// TIA Portal V15.1 export
// export: Created 2024-05-17T05:38:32.5503096Z, ExportSetting WithDefaults, DisplayName Totally Integrated Automation Portal, DisplayVersion V15.1 Update 5, DisplayName TIA Portal Openness, DisplayVersion V15.1 Update 5, DisplayName SINAMICS Startdrive Advanced, DisplayVersion V15.1, DisplayName G130, G150, S120, S150, SINAMICS MV, S210, DisplayVersion V15.1, DisplayName G110M, G120, G120C, G120D, G120P, DisplayVersion V15.1, DisplayName STEP 7 Professional, DisplayVersion V15.1 Update 5, DisplayName STEP 7 Safety, DisplayVersion V15.1, DisplayName WinCC Professional, DisplayVersion V15.1 Update 5, DisplayName SIMATIC Visualization Architect, DisplayVersion V15.1
FUNCTION_BLOCK "LMovFnc3Pos"   // FB2187, FBD
TITLE = LMovFnc3Pos
{ S7_Optimized_Access := 'TRUE' }
AUTHOR : VCC
FAMILY : Tooling
VERSION : 0.1
// =============================================================================
// This module will be used for the steering of a three Position movement.
// It will get the commands from different Modes, evaluate the status of the 
// Interlock and give the command to the Actuator or direct to simple outputs.
// =============================================================================
// stored: AutoNumber false, IsIECCheckEnabled false, IsRetainMemResEnabled false, MemoryReserve 100, SetENOAutomatically False, UDAEnableTagReadback false
   VAR_INPUT
      I_Pos1 { ExternalAccessible := 'False'; ExternalVisible := 'False'; ExternalWritable := 'False'} : Bool;   // Position Set detection or summary / Position 1 Detection
      I_Pos2 { ExternalAccessible := 'False'; ExternalVisible := 'False'; ExternalWritable := 'False'} : Bool;   // Position 2 Detection
      I_Pos3 { ExternalAccessible := 'False'; ExternalVisible := 'False'; ExternalWritable := 'False'} : Bool;   // Position Reset detection or summary / Position 3 Detection
      I_PBSet { ExternalAccessible := 'False'; ExternalVisible := 'False'; ExternalWritable := 'False'} : Bool;   // Push button for Set direction (used in manual with button OP panels )
      I_PBReset { ExternalAccessible := 'False'; ExternalVisible := 'False'; ExternalWritable := 'False'} : Bool;   // Push button for reset direcion (used in manual with pushbutton OP panels) / Push button for Reset direction (used in manual with Pushbutton OP panels)
      I_Pos1Begin { ExternalAccessible := 'False'; ExternalVisible := 'False'; ExternalWritable := 'False'} : Bool;   // Function Set begin selection / Function Pos1 begin selection
      I_Pos2Begin { ExternalAccessible := 'False'; ExternalVisible := 'False'; ExternalWritable := 'False'} : Bool;   // Function Set begin selection / Function Pos2 begin selection
      I_Pos3Begin { ExternalAccessible := 'False'; ExternalVisible := 'False'; ExternalWritable := 'False'} : Bool;   // Function Reset begin selection / Function Pos3 begin selection
      I_Pos1IntlkOK { ExternalAccessible := 'False'; ExternalVisible := 'False'; ExternalWritable := 'False'} : Bool;   // Set Interlock / Pos1 Interlock
      I_Pos2IntlkOK { ExternalAccessible := 'False'; ExternalVisible := 'False'; ExternalWritable := 'False'} : Bool;   // Set Interlock / Pos2 Interlock
      I_Pos3IntlkOK { ExternalAccessible := 'False'; ExternalVisible := 'False'; ExternalWritable := 'False'} : Bool;   // Reset Interlock / Pos3 Interlock
      I_MiddleReachedManSTOP { ExternalAccessible := 'False'; ExternalVisible := 'False'; ExternalWritable := 'False'} : Bool;   // Middle pos reached
      I_SafetyOk { ExternalAccessible := 'False'; ExternalVisible := 'False'; ExternalWritable := 'False'} : Bool;   // Safety Ok
      I_HardwareOk { ExternalAccessible := 'False'; ExternalVisible := 'False'; ExternalWritable := 'False'} : Bool;   // Safety Ok / Hardware Ok
   END_VAR
   VAR_OUTPUT
      O_CmdPos1 { ExternalAccessible := 'False'; ExternalVisible := 'False'; ExternalWritable := 'False'} : Bool;   // Command to activate Set movement / Command to Activate Pos1 movement
      O_CmdPos2 { ExternalAccessible := 'False'; ExternalVisible := 'False'; ExternalWritable := 'False'} : Bool;   // Command to activate Set movement / Command to Activate Pos2 movement
      O_CmdPos3 { ExternalAccessible := 'False'; ExternalVisible := 'False'; ExternalWritable := 'False'} : Bool;   // Command to activate Reset movement / Command to Activate Pos3 movement
      O_FuncRunning { ExternalAccessible := 'False'; ExternalVisible := 'False'; ExternalWritable := 'False'} : Bool;   // Signal that the function is running
      O_FuncBusyTM { ExternalAccessible := 'False'; ExternalVisible := 'False'; ExternalWritable := 'False'} : Bool;   // Memory Signal that the function is busy
      O_Pos1Finished { ExternalAccessible := 'False'; ExternalVisible := 'False'; ExternalWritable := 'False'} : Bool;   // Function Set finished to Master Sequencing / Function Pos1 finished to Master Sequencing
      O_Pos2Finished { ExternalAccessible := 'False'; ExternalVisible := 'False'; ExternalWritable := 'False'} : Bool;   // Function Set finished to Master Sequencing / Function Pos2 finished to Master Sequencing
      O_Pos3Finished { ExternalAccessible := 'False'; ExternalVisible := 'False'; ExternalWritable := 'False'} : Bool;   // Function Reset finished to Master Sequencing / Function Pos3 finished to Master Sequencing
      O_IntlkPos1Alm { ExternalAccessible := 'False'; ExternalVisible := 'False'; ExternalWritable := 'False'} : Bool;   // Alarm interlock Set / Alarm Interlock Pos1
      O_IntlkPos2Alm { ExternalAccessible := 'False'; ExternalVisible := 'False'; ExternalWritable := 'False'} : Bool;   // Alarm interlock Set / Alarm Interlock Pos2
      O_IntlkPos3Alm { ExternalAccessible := 'False'; ExternalVisible := 'False'; ExternalWritable := 'False'} : Bool;   // Alarm interlock Reset / Alarm Interlock Reset
      O_FuncIsSelInMan { ExternalAccessible := 'False'; ExternalVisible := 'False'; ExternalWritable := 'False'} : Bool;   // The function is selected in manual mode / The function is Selected in manual Mode
      O_LED { ExternalAccessible := 'False'; ExternalVisible := 'False'; ExternalWritable := 'False'} : Bool;   // LED - Indication
      O_AlarmABCondition { ExternalAccessible := 'False'; ExternalVisible := 'False'; ExternalWritable := 'False'} : Bool;   // Alarms AB condition / Alarm AB Condition
   END_VAR
   VAR_IN_OUT
      IO_Modes : "Modes";   // Modes
      H_HMI : "H_HMI";   // Animation
      H_MovFnc3Pos : "H_MovFnc3Pos";   // Animation
      H_FncSelInHMI { ExternalAccessible := 'False'; ExternalVisible := 'False'; ExternalWritable := 'False'} : Bool;   // This function is selected to run from HMI / This function is Selected to run from HMI
      C_AlarmResetUsed { ExternalAccessible := 'False'; ExternalVisible := 'False'; ExternalWritable := 'False'} : Bool;   // If true, the alrms will be stored untill reseted / If TRUE The Alarms will be stored untill Reseted
      C_EnableMemBegin { ExternalAccessible := 'False'; ExternalVisible := 'False'; ExternalWritable := 'False'} : Bool;   // Enable memory Begin (Command request is memorised until pos reached) / Enable memory Begin (Command Request is memorised until pos reached)
      C_EnIntlkAlm { ExternalAccessible := 'False'; ExternalVisible := 'False'; ExternalWritable := 'False'} : Bool := TRUE;   // Enable Interlock Alarm
      C_SetReset { ExternalAccessible := 'False'; ExternalVisible := 'False'; ExternalWritable := 'False'} : Bool;   // Enable Set Reset Functionality ( If enabled output is kept until the Cmd direction is changed )
      C_ForceManual { ExternalAccessible := 'False'; ExternalVisible := 'False'; ExternalWritable := 'False'} : Bool := FALSE;   // Force Manual
   END_VAR
   VAR
      ResetAlarm { ExternalAccessible := 'False'; ExternalVisible := 'False'; ExternalWritable := 'False'} : Bool;   // Reset Alarm Memory
      CmdPos1Request { ExternalAccessible := 'False'; ExternalVisible := 'False'; ExternalWritable := 'False'} : Bool;   // Set Command request to activate the interlock / Pos1 Command Request to Activate the Interlock
      CmdPos2Request { ExternalAccessible := 'False'; ExternalVisible := 'False'; ExternalWritable := 'False'} : Bool;   // Set Command request to activate the interlock / Pos1 Command Request to Activate the Interlock
      CmdPos3Request { ExternalAccessible := 'False'; ExternalVisible := 'False'; ExternalWritable := 'False'} : Bool;   // Reset Command request to activate the interlock / Pos3 Command Request to Activate the Interlock
      EdgeStopDetPos1 { ExternalAccessible := 'False'; ExternalVisible := 'False'; ExternalWritable := 'False'} : Bool;   // Edge on stop detection to be abble to go over it in force manual
      EdgeStopDetPos2 { ExternalAccessible := 'False'; ExternalVisible := 'False'; ExternalWritable := 'False'} : Bool;   // Edge on stop detection to be abble to go over it in force manual
      EdgeStopDetPos3 { ExternalAccessible := 'False'; ExternalVisible := 'False'; ExternalWritable := 'False'} : Bool;   // Edge on stop detection to be abble to go over it in force manual
      IntlkPos1Alm { ExternalAccessible := 'False'; ExternalVisible := 'False'; ExternalWritable := 'False'} : Bool;   // Alarm interlock Set / Alarm Interlock Pos1
      IntlkPos2Alm { ExternalAccessible := 'False'; ExternalVisible := 'False'; ExternalWritable := 'False'} : Bool;   // Alarm interlock Set / Alarm Interlock Pos2
      IntlkPos3Alm { ExternalAccessible := 'False'; ExternalVisible := 'False'; ExternalWritable := 'False'} : Bool;   // Alarm interlock Reset / Alarm Interlock Reset
      CmdPos1 { ExternalAccessible := 'False'; ExternalVisible := 'False'; ExternalWritable := 'False'} : Bool;   // Command to activate Set movement / Command to Activate Pos1 movement
      CmdPos2 { ExternalAccessible := 'False'; ExternalVisible := 'False'; ExternalWritable := 'False'} : Bool;   // Command to activate Set movement / Command to Activate Pos2 movement
      CmdPos3 { ExternalAccessible := 'False'; ExternalVisible := 'False'; ExternalWritable := 'False'} : Bool;   // Command to activate Reset movement / Command to Activate Pos3 movement
      IntlkPos1AlmCond { ExternalAccessible := 'False'; ExternalVisible := 'False'; ExternalWritable := 'False'} : Bool;   // Alarm interlock Set condition / Alarm Interlock Pos1 condition
      IntlkPos2AlmCond { ExternalAccessible := 'False'; ExternalVisible := 'False'; ExternalWritable := 'False'} : Bool;   // Alarm interlock Set condition / Alarm Interlock Pos2 condition
      IntlkPos3AlmCond { ExternalAccessible := 'False'; ExternalVisible := 'False'; ExternalWritable := 'False'} : Bool;   // Alarm interlock Reset condition / Alarm Interlock Pos3 condition
      FuncRunning { ExternalAccessible := 'False'; ExternalVisible := 'False'; ExternalWritable := 'False'} : Bool;   // Function is running
      LampTest { ExternalAccessible := 'False'; ExternalVisible := 'False'; ExternalWritable := 'False'} : Bool;   // Lamp test
      LampTestSteady { ExternalAccessible := 'False'; ExternalVisible := 'False'; ExternalWritable := 'False'} : Bool;   // Lamp test always on from mode of station / Lamp test always on from Mode of station
      FuncBusyTM { ExternalAccessible := 'False'; ExternalVisible := 'False'; ExternalWritable := 'False'} : Bool;   // Memory Signal that the function is busy
      AlarmTimer { ExternalAccessible := 'False'; ExternalVisible := 'False'; ExternalWritable := 'False'} : "LTimer";
      AlmFilterResult { ExternalAccessible := 'False'; ExternalVisible := 'False'; ExternalWritable := 'False'} : Bool;
   END_VAR
   VAR_TEMP   // added for the SCL form of the ladder/FBD networks
      _w1 : Bool;
   END_VAR
BEGIN

REGION Network 1: **** 2.2 - Alarms - Alarm Generation **** Alarm Filter
   // Alarm Filter
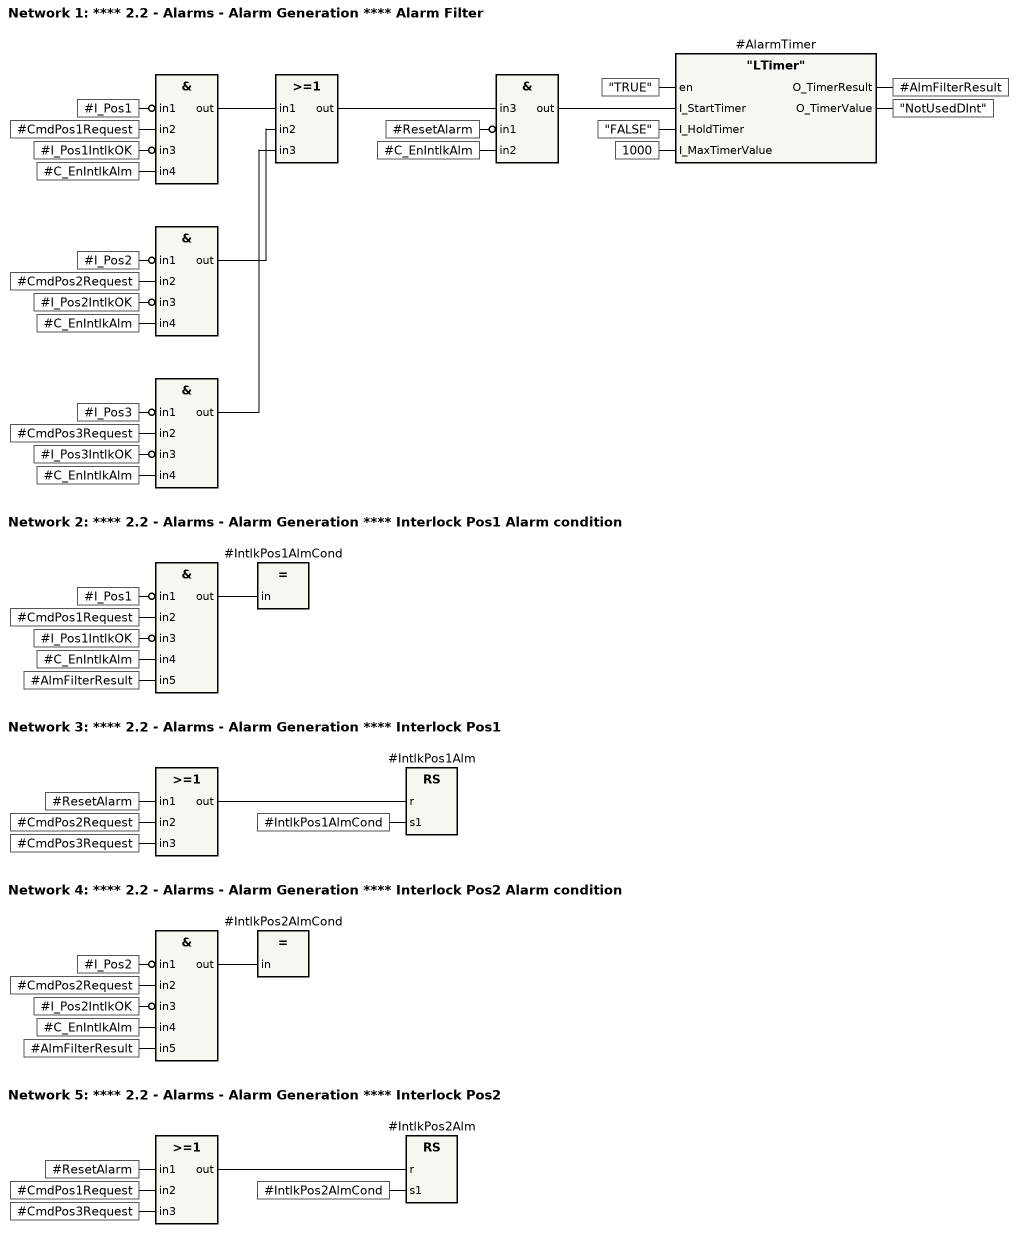
   IF "TRUE" THEN
       #AlarmTimer(I_StartTimer := ((NOT #I_Pos1 AND #CmdPos1Request AND NOT #I_Pos1IntlkOK AND #C_EnIntlkAlm) OR (NOT #I_Pos2 AND #CmdPos2Request AND NOT #I_Pos2IntlkOK AND #C_EnIntlkAlm) OR (NOT #I_Pos3 AND #CmdPos3Request AND NOT #I_Pos3IntlkOK AND #C_EnIntlkAlm)) AND NOT #ResetAlarm AND #C_EnIntlkAlm,   // "LTimer"
                   I_HoldTimer := "FALSE",
                   I_MaxTimerValue := 1000,
                   O_TimerResult => #AlmFilterResult,
                   O_TimerValue => "NotUsedDInt");
   END_IF;
END_REGION

REGION Network 2: **** 2.2 - Alarms - Alarm Generation **** Interlock Pos1 Alarm condition
   // Interlock Pos1 Alarm condition
   #IntlkPos1AlmCond := NOT #I_Pos1 AND #CmdPos1Request AND NOT #I_Pos1IntlkOK AND #C_EnIntlkAlm AND #AlmFilterResult;
END_REGION

REGION Network 3: **** 2.2 - Alarms - Alarm Generation **** Interlock Pos1
   // Interlock Pos1
   IF #ResetAlarm OR #CmdPos2Request OR #CmdPos3Request THEN
       #IntlkPos1Alm := FALSE;   // RS flip-flop
   END_IF;
   IF #IntlkPos1AlmCond THEN #IntlkPos1Alm := TRUE; END_IF;
END_REGION

REGION Network 4: **** 2.2 - Alarms - Alarm Generation **** Interlock Pos2 Alarm condition
   // Interlock Pos2 Alarm condition
   #IntlkPos2AlmCond := NOT #I_Pos2 AND #CmdPos2Request AND NOT #I_Pos2IntlkOK AND #C_EnIntlkAlm AND #AlmFilterResult;
END_REGION

REGION Network 5: **** 2.2 - Alarms - Alarm Generation **** Interlock Pos2
   // Interlock Pos2
   IF #ResetAlarm OR #CmdPos1Request OR #CmdPos3Request THEN
       #IntlkPos2Alm := FALSE;   // RS flip-flop
   END_IF;
   IF #IntlkPos2AlmCond THEN #IntlkPos2Alm := TRUE; END_IF;
END_REGION

REGION Network 6: **** 2.2 - Alarms - Alarm Generation **** Interlock Pos3 Alarm condition
   // Interlock Pos3 Alarm condition
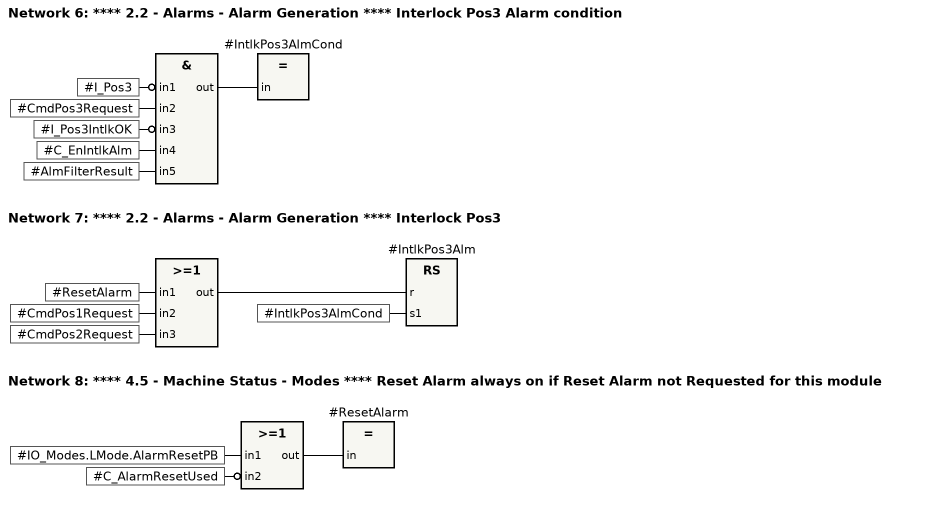
   #IntlkPos3AlmCond := NOT #I_Pos3 AND #CmdPos3Request AND NOT #I_Pos3IntlkOK AND #C_EnIntlkAlm AND #AlmFilterResult;
END_REGION

REGION Network 7: **** 2.2 - Alarms - Alarm Generation **** Interlock Pos3
   // Interlock Pos3
   IF #ResetAlarm OR #CmdPos1Request OR #CmdPos2Request THEN
       #IntlkPos3Alm := FALSE;   // RS flip-flop
   END_IF;
   IF #IntlkPos3AlmCond THEN #IntlkPos3Alm := TRUE; END_IF;
END_REGION

REGION Network 8: **** 4.5 - Machine Status - Modes **** Reset Alarm always on if Reset Alarm not Requested for this module
   // Reset Alarm always on if Reset Alarm not Requested for this module
   #ResetAlarm := #IO_Modes.LMode.AlarmResetPB OR NOT #C_AlarmResetUsed;
END_REGION

REGION Network 9: **** 4.6 - Machine Status - Indication **** Icon Animation
   // Icon Animation
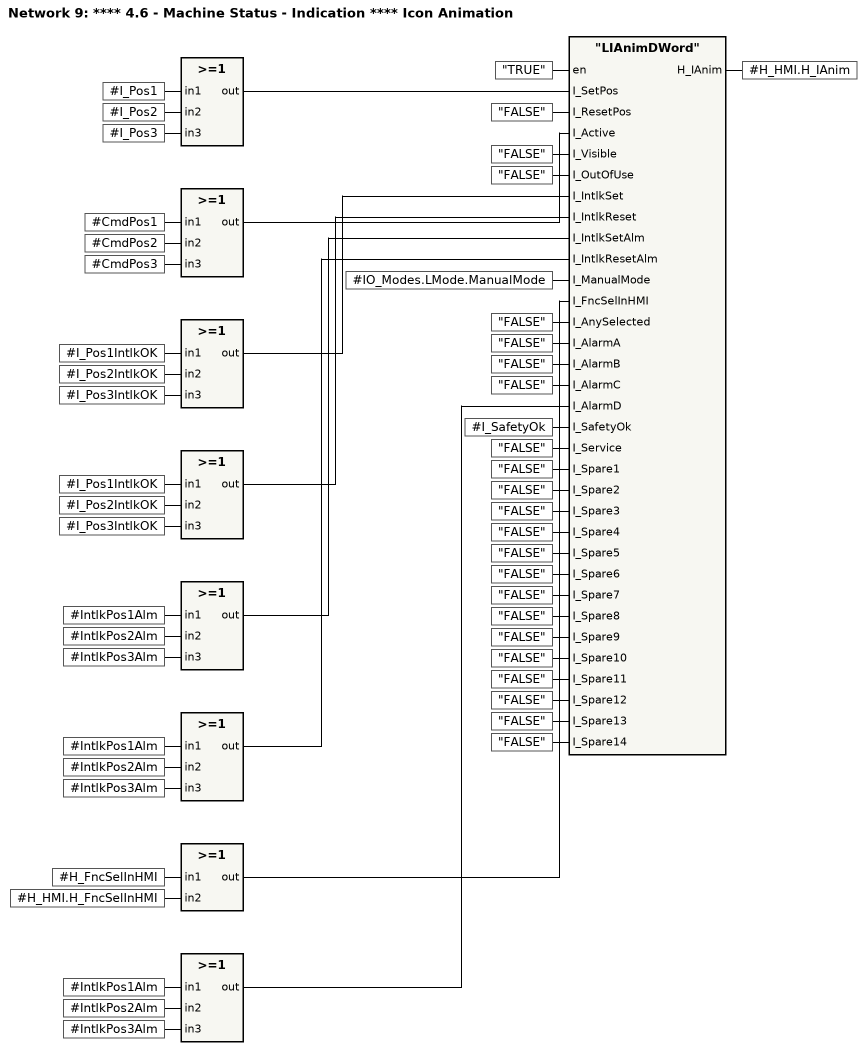
   IF "TRUE" THEN
       "LIAnimDWord"(I_SetPos := #I_Pos1 OR #I_Pos2 OR #I_Pos3,
                     I_ResetPos := "FALSE",
                     I_Active := #CmdPos1 OR #CmdPos2 OR #CmdPos3,
                     I_Visible := "FALSE",
                     I_OutOfUse := "FALSE",
                     I_IntlkSet := #I_Pos1IntlkOK OR #I_Pos2IntlkOK OR #I_Pos3IntlkOK,
                     I_IntlkReset := #I_Pos1IntlkOK OR #I_Pos2IntlkOK OR #I_Pos3IntlkOK,
                     I_IntlkSetAlm := #IntlkPos1Alm OR #IntlkPos2Alm OR #IntlkPos3Alm,
                     I_IntlkResetAlm := #IntlkPos1Alm OR #IntlkPos2Alm OR #IntlkPos3Alm,
                     I_ManualMode := #IO_Modes.LMode.ManualMode,
                     I_FncSelInHMI := #H_FncSelInHMI OR #H_HMI.H_FncSelInHMI,
                     I_AnySelected := "FALSE",
                     I_AlarmA := "FALSE",
                     I_AlarmB := "FALSE",
                     I_AlarmC := "FALSE",
                     I_AlarmD := #IntlkPos1Alm OR #IntlkPos2Alm OR #IntlkPos3Alm,
                     I_SafetyOk := #I_SafetyOk,
                     I_Service := "FALSE",
                     I_Spare1 := "FALSE",
                     I_Spare2 := "FALSE",
                     I_Spare3 := "FALSE",
                     I_Spare4 := "FALSE",
                     I_Spare5 := "FALSE",
                     I_Spare6 := "FALSE",
                     I_Spare7 := "FALSE",
                     I_Spare8 := "FALSE",
                     I_Spare9 := "FALSE",
                     I_Spare10 := "FALSE",
                     I_Spare11 := "FALSE",
                     I_Spare12 := "FALSE",
                     I_Spare13 := "FALSE",
                     I_Spare14 := "FALSE",
                     H_IAnim => #H_HMI.H_IAnim);
   END_IF;
END_REGION

REGION Network 10: **** 4.6 - Machine Status - Indication **** Animation
   // Animation
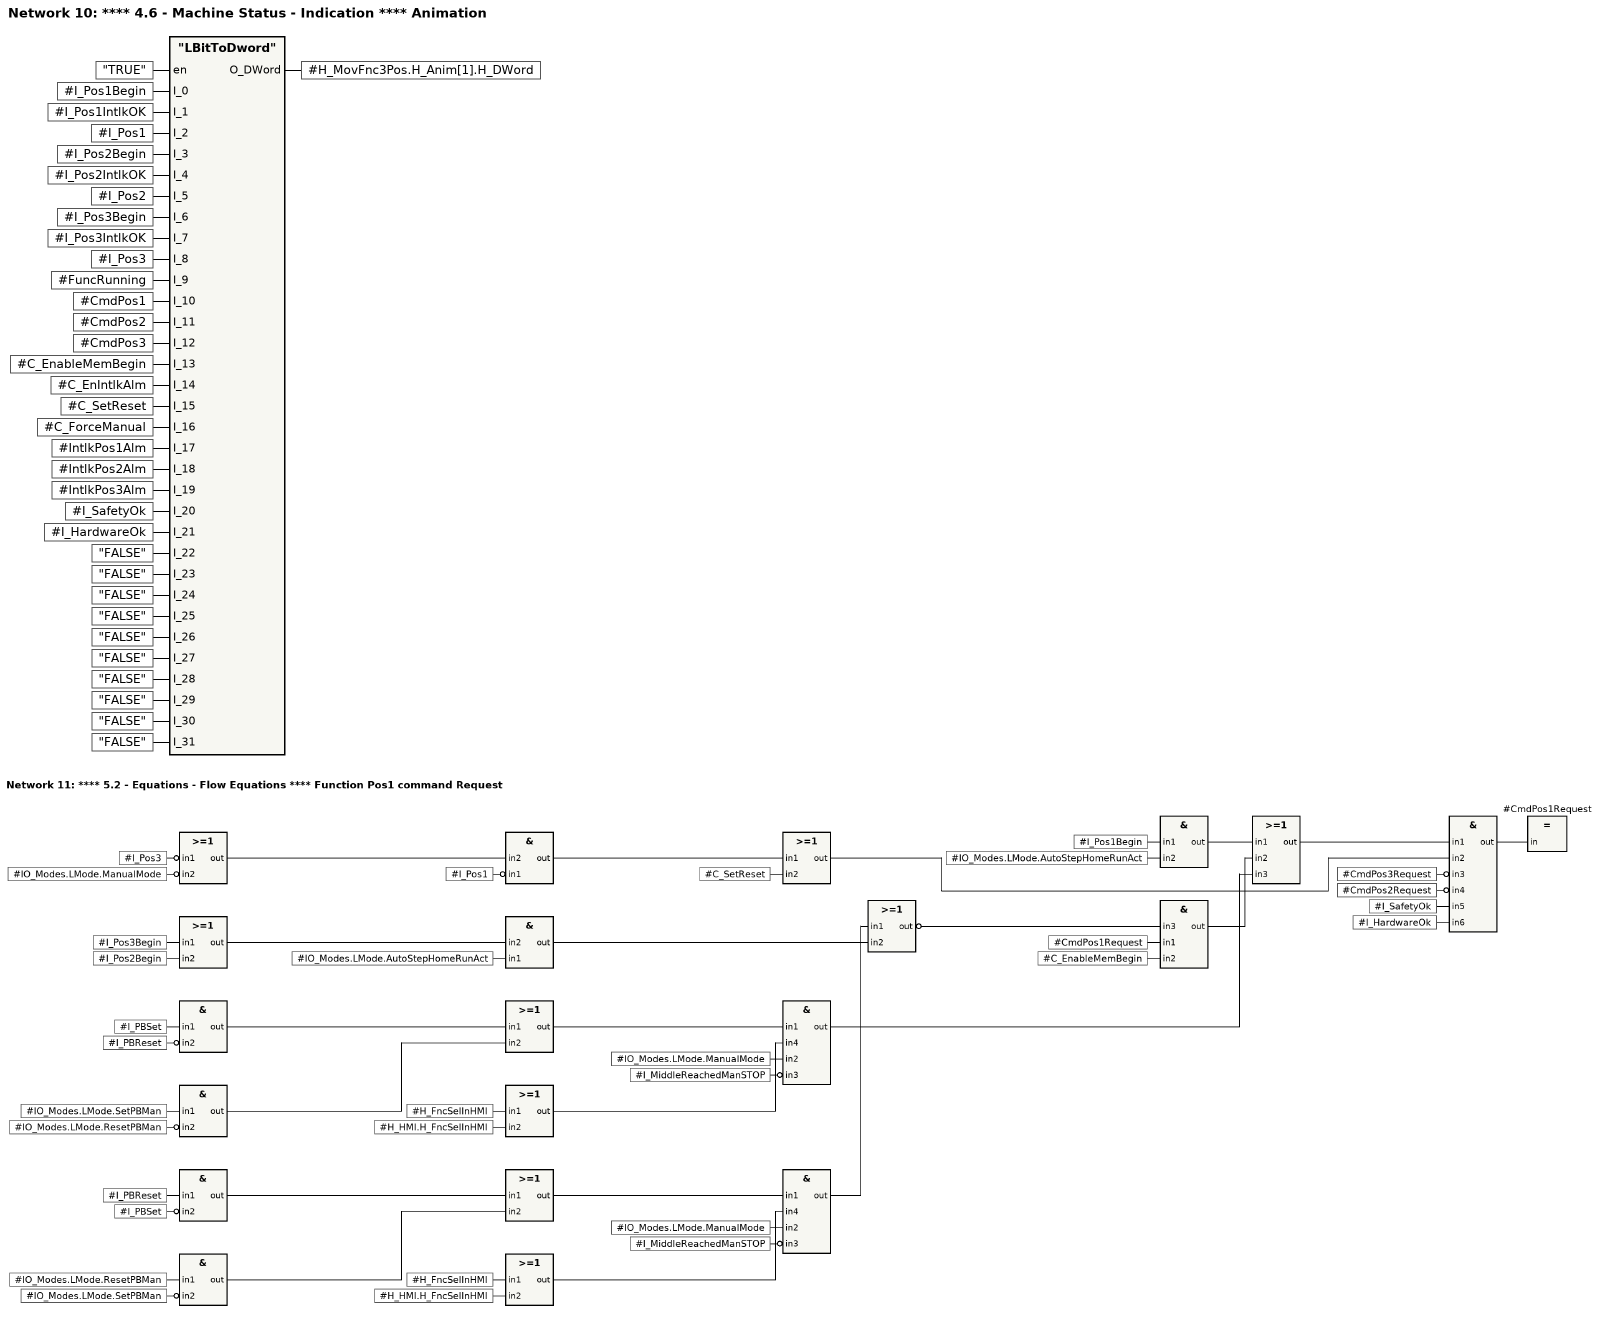
   IF "TRUE" THEN
       "LBitToDword"(I_0 := #I_Pos1Begin,
                     I_1 := #I_Pos1IntlkOK,
                     I_2 := #I_Pos1,
                     I_3 := #I_Pos2Begin,
                     I_4 := #I_Pos2IntlkOK,
                     I_5 := #I_Pos2,
                     I_6 := #I_Pos3Begin,
                     I_7 := #I_Pos3IntlkOK,
                     I_8 := #I_Pos3,
                     I_9 := #FuncRunning,
                     I_10 := #CmdPos1,
                     I_11 := #CmdPos2,
                     I_12 := #CmdPos3,
                     I_13 := #C_EnableMemBegin,
                     I_14 := #C_EnIntlkAlm,
                     I_15 := #C_SetReset,
                     I_16 := #C_ForceManual,
                     I_17 := #IntlkPos1Alm,
                     I_18 := #IntlkPos2Alm,
                     I_19 := #IntlkPos3Alm,
                     I_20 := #I_SafetyOk,
                     I_21 := #I_HardwareOk,
                     I_22 := "FALSE",
                     I_23 := "FALSE",
                     I_24 := "FALSE",
                     I_25 := "FALSE",
                     I_26 := "FALSE",
                     I_27 := "FALSE",
                     I_28 := "FALSE",
                     I_29 := "FALSE",
                     I_30 := "FALSE",
                     I_31 := "FALSE",
                     O_DWord => #H_MovFnc3Pos.H_Anim[1].H_DWord);
   END_IF;
END_REGION

REGION Network 11: **** 5.2 - Equations - Flow Equations **** Function Pos1 command Request
   // Function Pos1 command Request
   #CmdPos1Request := ((#I_Pos1Begin AND #IO_Modes.LMode.AutoStepHomeRunAct) OR (NOT ((((#I_PBReset AND NOT #I_PBSet) OR (#IO_Modes.LMode.ResetPBMan AND NOT #IO_Modes.LMode.SetPBMan)) AND (#H_FncSelInHMI OR #H_HMI.H_FncSelInHMI) AND #IO_Modes.LMode.ManualMode AND NOT #I_MiddleReachedManSTOP) OR ((#I_Pos3Begin OR #I_Pos2Begin) AND #IO_Modes.LMode.AutoStepHomeRunAct)) AND #CmdPos1Request AND #C_EnableMemBegin) OR (((#I_PBSet AND NOT #I_PBReset) OR (#IO_Modes.LMode.SetPBMan AND NOT #IO_Modes.LMode.ResetPBMan)) AND (#H_FncSelInHMI OR #H_HMI.H_FncSelInHMI) AND #IO_Modes.LMode.ManualMode AND NOT #I_MiddleReachedManSTOP)) AND (((NOT #I_Pos3 OR NOT #IO_Modes.LMode.ManualMode) AND NOT #I_Pos1) OR #C_SetReset) AND NOT #CmdPos3Request AND NOT #CmdPos2Request AND #I_SafetyOk AND #I_HardwareOk;
END_REGION

REGION Network 12: **** 5.2 - Equations - Flow Equations **** Function Pos2 command Request
   // Function Pos2 command Request
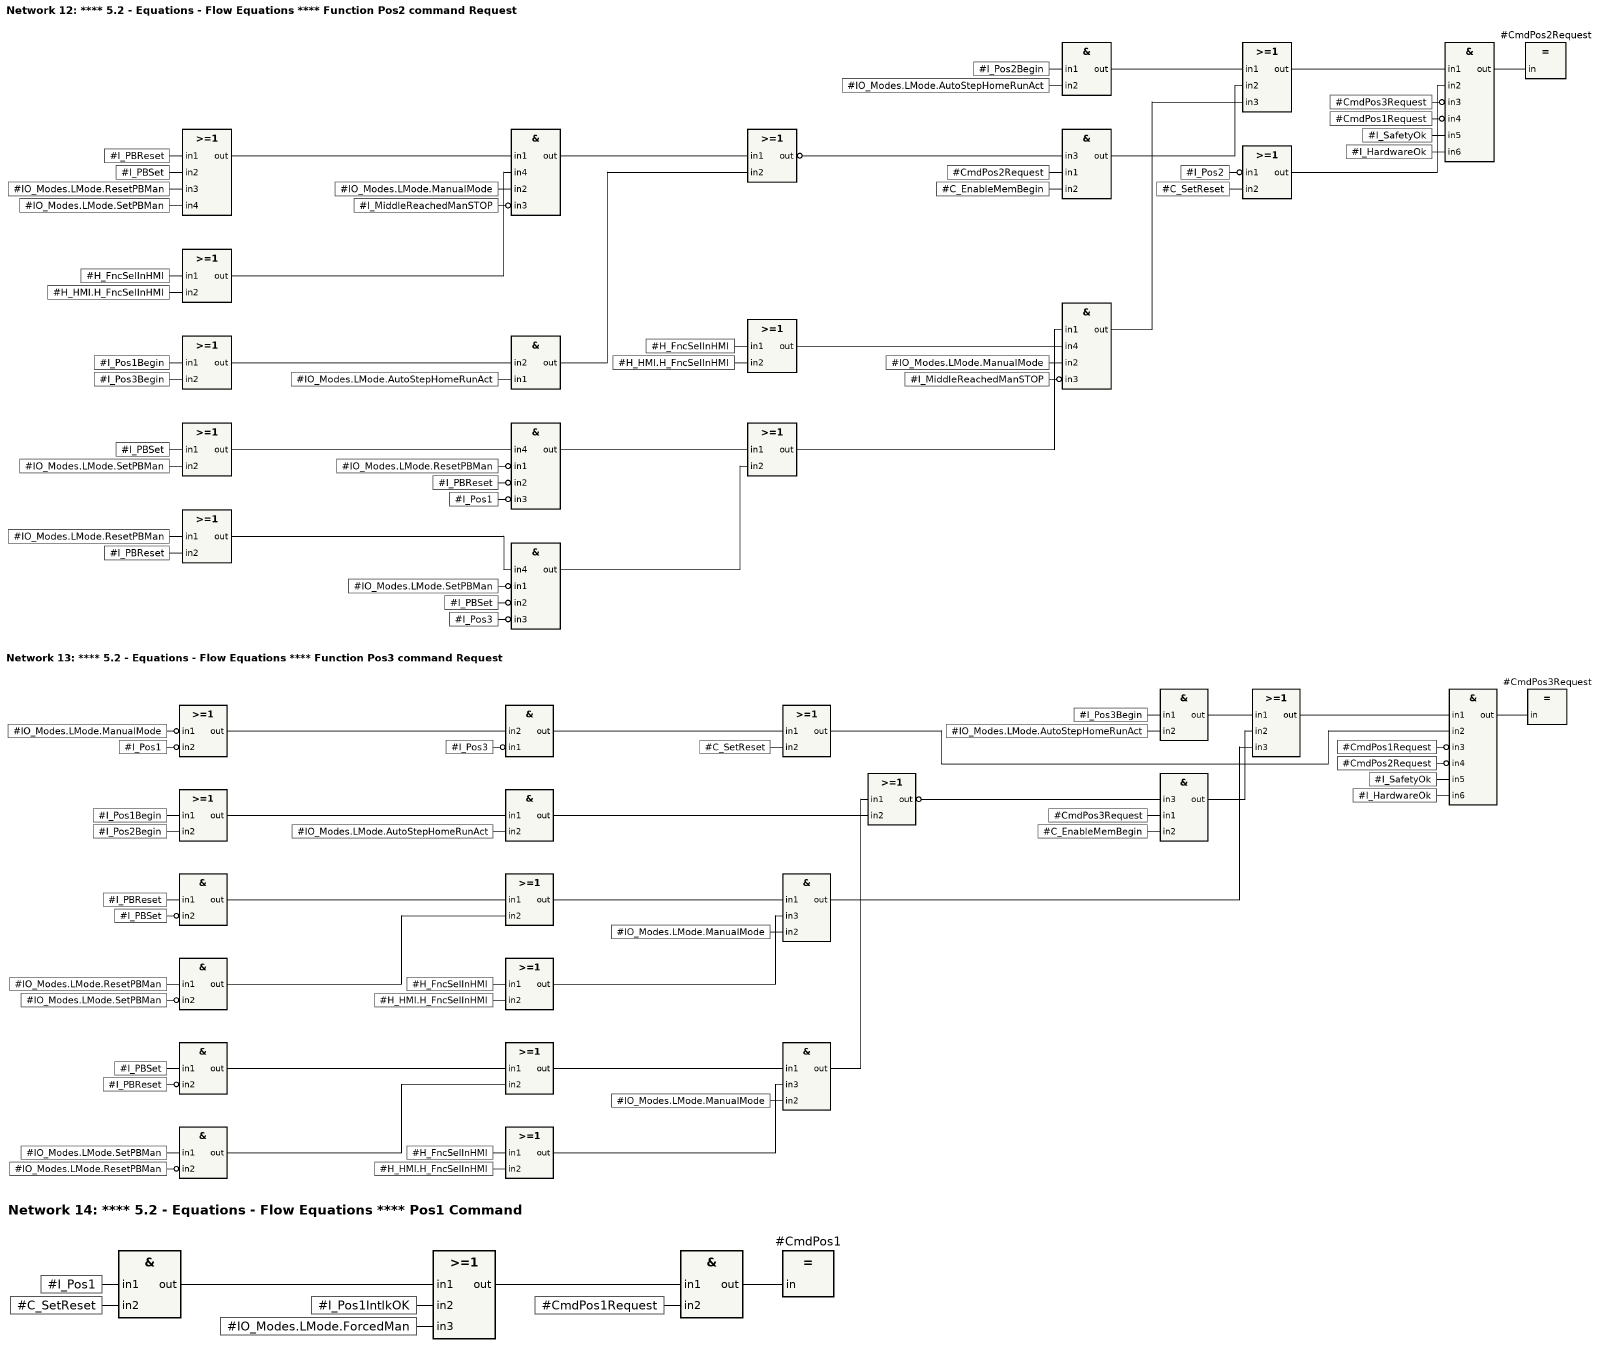
   #CmdPos2Request := ((#I_Pos2Begin AND #IO_Modes.LMode.AutoStepHomeRunAct) OR (NOT (((#I_PBReset OR #I_PBSet OR #IO_Modes.LMode.ResetPBMan OR #IO_Modes.LMode.SetPBMan) AND (#H_FncSelInHMI OR #H_HMI.H_FncSelInHMI) AND #IO_Modes.LMode.ManualMode AND NOT #I_MiddleReachedManSTOP) OR ((#I_Pos1Begin OR #I_Pos3Begin) AND #IO_Modes.LMode.AutoStepHomeRunAct)) AND #CmdPos2Request AND #C_EnableMemBegin) OR ((((#I_PBSet OR #IO_Modes.LMode.SetPBMan) AND NOT #IO_Modes.LMode.ResetPBMan AND NOT #I_PBReset AND NOT #I_Pos1) OR ((#IO_Modes.LMode.ResetPBMan OR #I_PBReset) AND NOT #IO_Modes.LMode.SetPBMan AND NOT #I_PBSet AND NOT #I_Pos3)) AND (#H_FncSelInHMI OR #H_HMI.H_FncSelInHMI) AND #IO_Modes.LMode.ManualMode AND NOT #I_MiddleReachedManSTOP)) AND (NOT #I_Pos2 OR #C_SetReset) AND NOT #CmdPos3Request AND NOT #CmdPos1Request AND #I_SafetyOk AND #I_HardwareOk;
END_REGION

REGION Network 13: **** 5.2 - Equations - Flow Equations **** Function Pos3 command Request
   // Function Pos3 command Request
   #CmdPos3Request := ((#I_Pos3Begin AND #IO_Modes.LMode.AutoStepHomeRunAct) OR (NOT ((((#I_PBSet AND NOT #I_PBReset) OR (#IO_Modes.LMode.SetPBMan AND NOT #IO_Modes.LMode.ResetPBMan)) AND (#H_FncSelInHMI OR #H_HMI.H_FncSelInHMI) AND #IO_Modes.LMode.ManualMode) OR ((#I_Pos1Begin OR #I_Pos2Begin) AND #IO_Modes.LMode.AutoStepHomeRunAct)) AND #CmdPos3Request AND #C_EnableMemBegin) OR (((#I_PBReset AND NOT #I_PBSet) OR (#IO_Modes.LMode.ResetPBMan AND NOT #IO_Modes.LMode.SetPBMan)) AND (#H_FncSelInHMI OR #H_HMI.H_FncSelInHMI) AND #IO_Modes.LMode.ManualMode)) AND (((NOT #IO_Modes.LMode.ManualMode OR NOT #I_Pos1) AND NOT #I_Pos3) OR #C_SetReset) AND NOT #CmdPos1Request AND NOT #CmdPos2Request AND #I_SafetyOk AND #I_HardwareOk;
END_REGION

REGION Network 14: **** 5.2 - Equations - Flow Equations **** Pos1 Command
   // Pos1 Command
   #CmdPos1 := ((#I_Pos1 AND #C_SetReset) OR #I_Pos1IntlkOK OR #IO_Modes.LMode.ForcedMan) AND #CmdPos1Request;
END_REGION

REGION Network 15: **** 5.2 - Equations - Flow Equations **** Pos2 Command
   // Pos2 Command
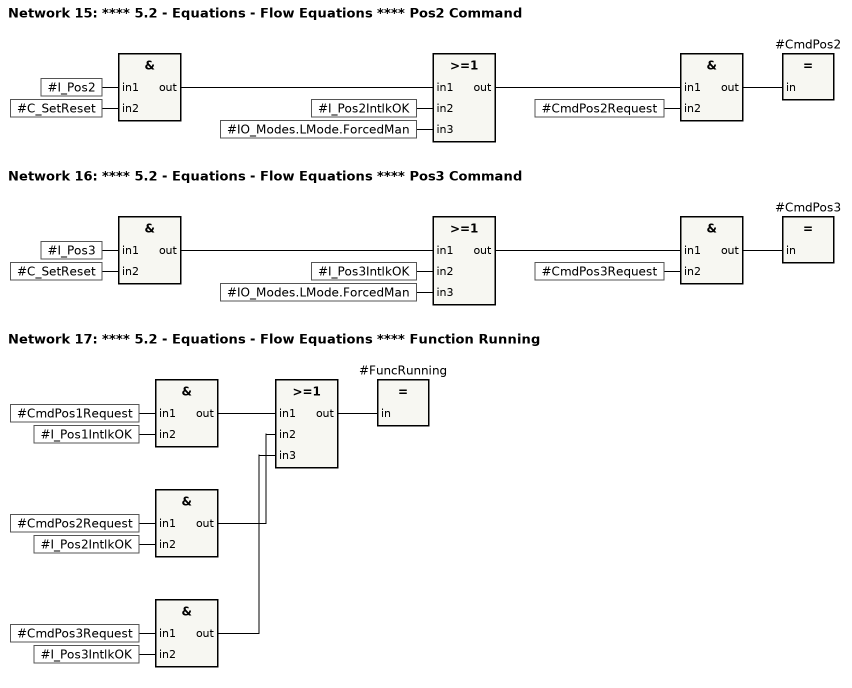
   #CmdPos2 := ((#I_Pos2 AND #C_SetReset) OR #I_Pos2IntlkOK OR #IO_Modes.LMode.ForcedMan) AND #CmdPos2Request;
END_REGION

REGION Network 16: **** 5.2 - Equations - Flow Equations **** Pos3 Command
   // Pos3 Command
   #CmdPos3 := ((#I_Pos3 AND #C_SetReset) OR #I_Pos3IntlkOK OR #IO_Modes.LMode.ForcedMan) AND #CmdPos3Request;
END_REGION

REGION Network 17: **** 5.2 - Equations - Flow Equations **** Function Running
   // Function Running
   #FuncRunning := (#CmdPos1Request AND #I_Pos1IntlkOK) OR (#CmdPos2Request AND #I_Pos2IntlkOK) OR (#CmdPos3Request AND #I_Pos3IntlkOK);
END_REGION

REGION Network 18: **** 5.2 - Equations - Flow Equations **** Function Running Memory
   // Function Running Memory
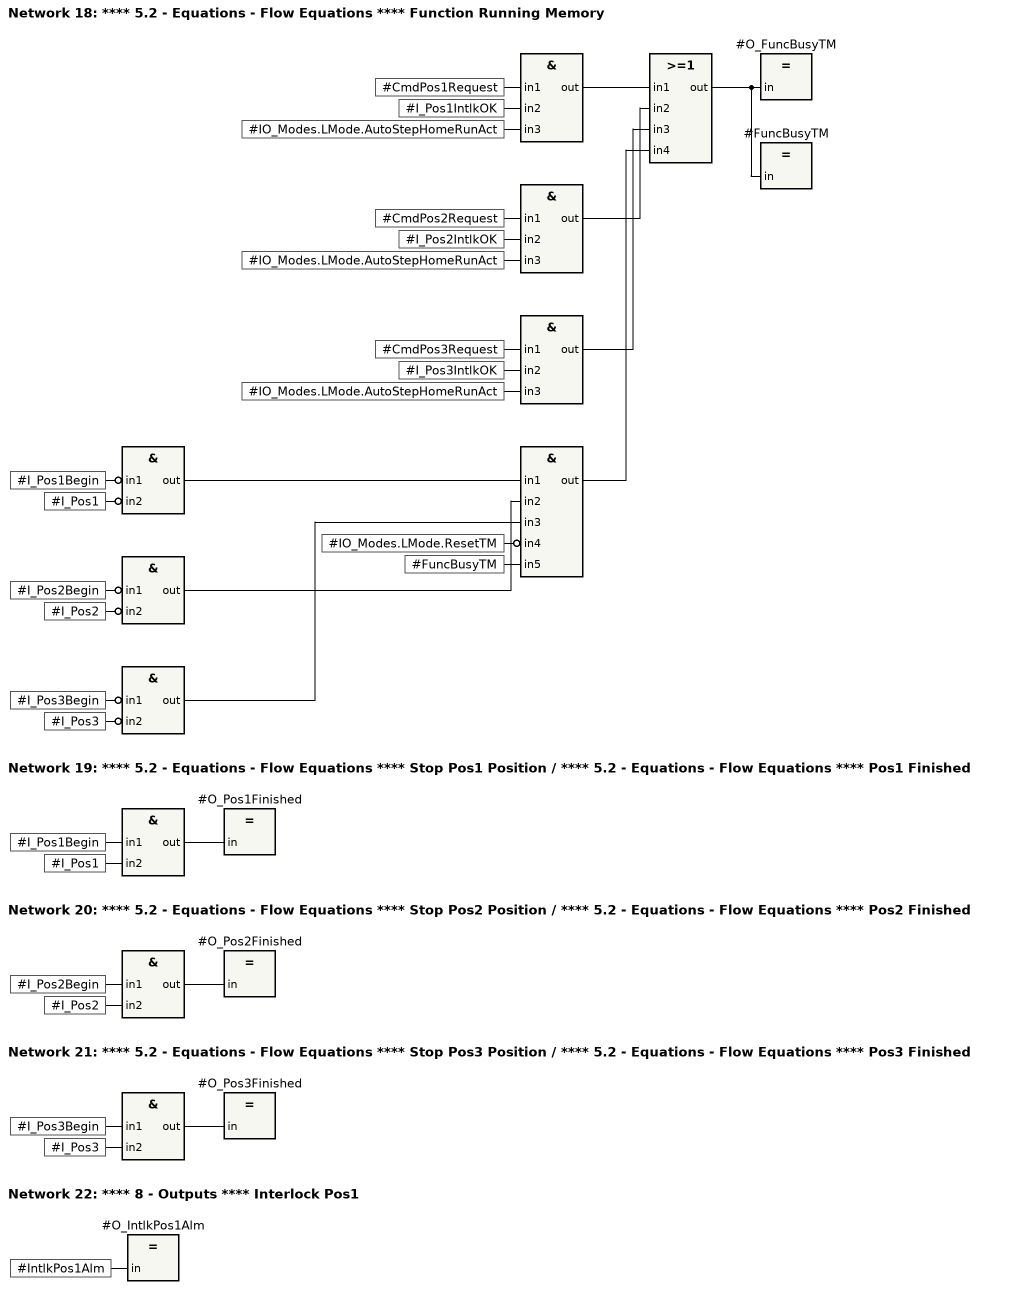
   #O_FuncBusyTM := (#CmdPos1Request AND #I_Pos1IntlkOK AND #IO_Modes.LMode.AutoStepHomeRunAct) OR (#CmdPos2Request AND #I_Pos2IntlkOK AND #IO_Modes.LMode.AutoStepHomeRunAct) OR (#CmdPos3Request AND #I_Pos3IntlkOK AND #IO_Modes.LMode.AutoStepHomeRunAct) OR (NOT #I_Pos1Begin AND NOT #I_Pos1 AND NOT #I_Pos2Begin AND NOT #I_Pos2 AND NOT #I_Pos3Begin AND NOT #I_Pos3 AND NOT #IO_Modes.LMode.ResetTM AND #FuncBusyTM);
   #FuncBusyTM := #O_FuncBusyTM;
END_REGION

REGION Network 19: **** 5.2 - Equations - Flow Equations **** Stop Pos1 Position / **** 5.2 - Equations - Flow Equations **** Pos1 Finished
   // Interlock Pos1
   #O_Pos1Finished := #I_Pos1Begin AND #I_Pos1;
END_REGION

REGION Network 20: **** 5.2 - Equations - Flow Equations **** Stop Pos2 Position / **** 5.2 - Equations - Flow Equations **** Pos2 Finished
   // Interlock Pos2
   #O_Pos2Finished := #I_Pos2Begin AND #I_Pos2;
END_REGION

REGION Network 21: **** 5.2 - Equations - Flow Equations **** Stop Pos3 Position / **** 5.2 - Equations - Flow Equations **** Pos3 Finished
   // Stop Pos3 Position
   #O_Pos3Finished := #I_Pos3Begin AND #I_Pos3;
END_REGION

REGION Network 22: **** 8 - Outputs **** Interlock Pos1
   // Interlock Pos1
   #O_IntlkPos1Alm := #IntlkPos1Alm;
END_REGION

REGION Network 23: **** 8 - Outputs **** Interlock Pos2
   // Interlock Pos2
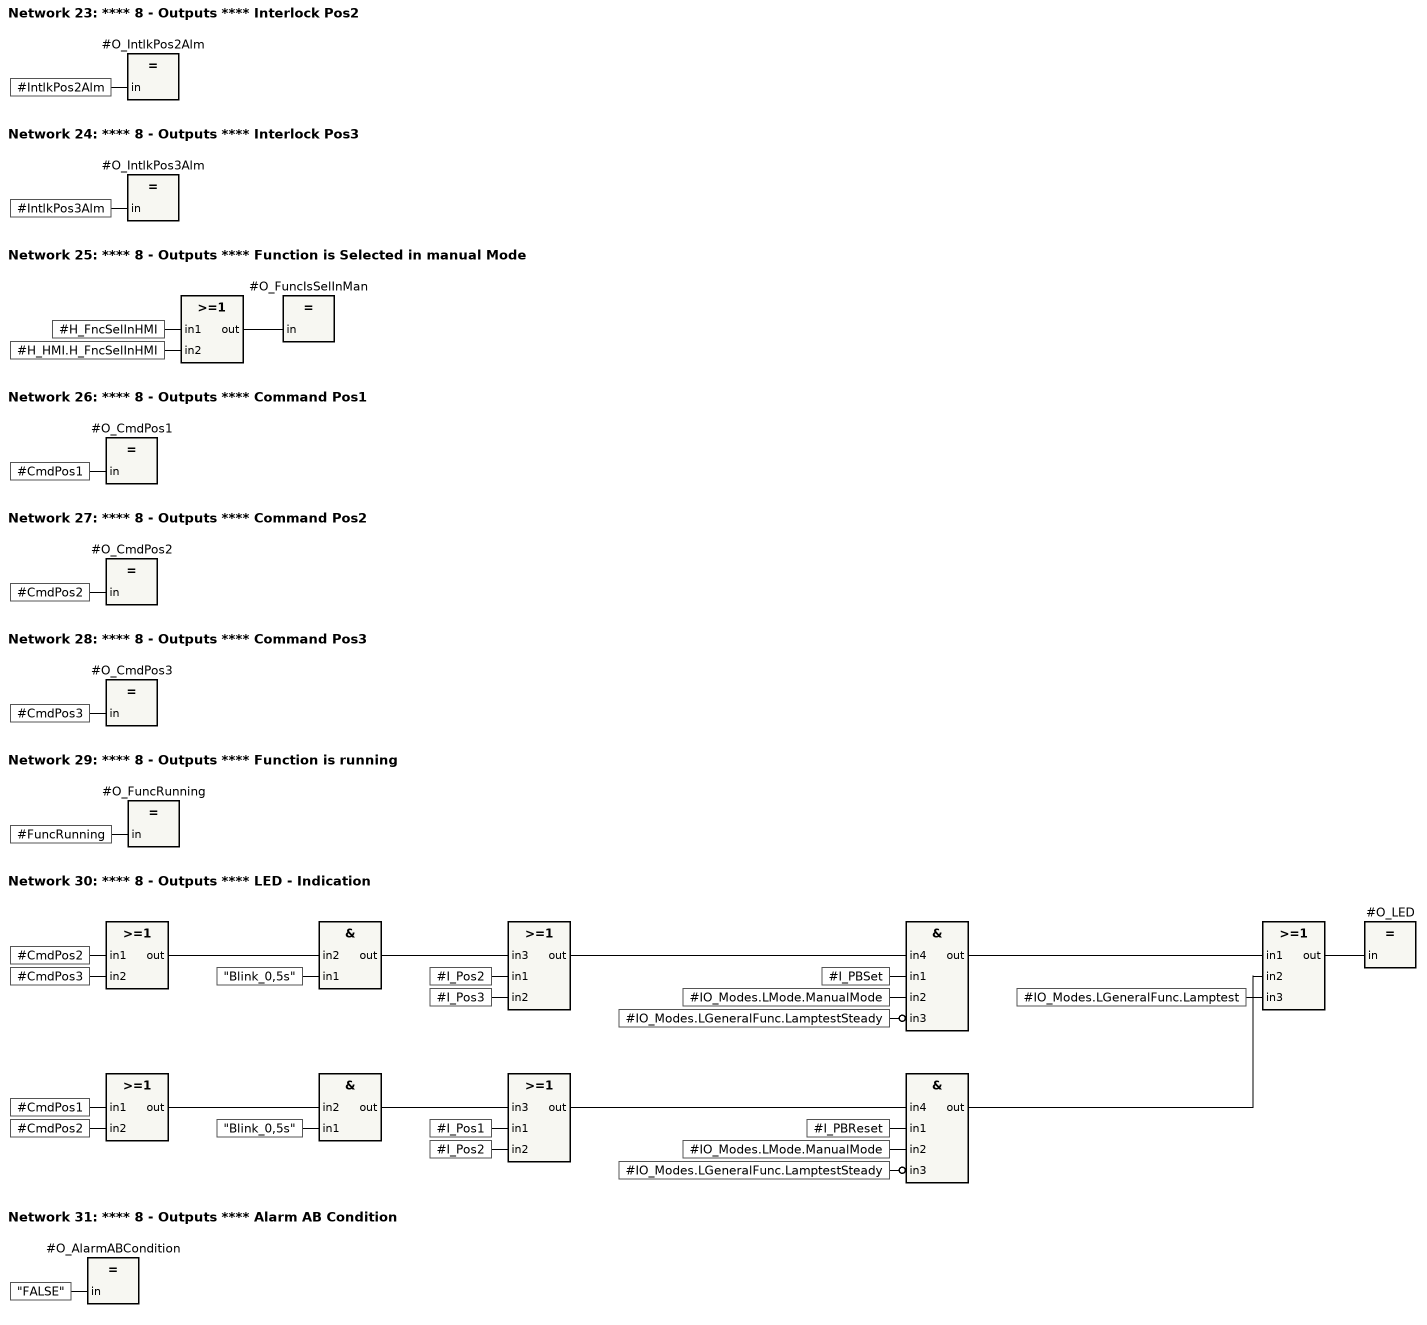
   #O_IntlkPos2Alm := #IntlkPos2Alm;
END_REGION

REGION Network 24: **** 8 - Outputs **** Interlock Pos3
   // Interlock Pos3
   #O_IntlkPos3Alm := #IntlkPos3Alm;
END_REGION

REGION Network 25: **** 8 - Outputs **** Function is Selected in manual Mode
   // Function is Selected in manual Mode
   #O_FuncIsSelInMan := #H_FncSelInHMI OR #H_HMI.H_FncSelInHMI;
END_REGION

REGION Network 26: **** 8 - Outputs **** Command Pos1
   // Command Pos1
   #O_CmdPos1 := #CmdPos1;
END_REGION

REGION Network 27: **** 8 - Outputs **** Command Pos2
   // Command Pos2
   #O_CmdPos2 := #CmdPos2;
END_REGION

REGION Network 28: **** 8 - Outputs **** Command Pos3
   // Command Pos3
   #O_CmdPos3 := #CmdPos3;
END_REGION

REGION Network 29: **** 8 - Outputs **** Function is running
   // Function is running
   #O_FuncRunning := #FuncRunning;
END_REGION

REGION Network 30: **** 8 - Outputs **** LED - Indication
   // LED - Indication
   #O_LED := ((((#CmdPos2 OR #CmdPos3) AND "Blink_0,5s") OR #I_Pos2 OR #I_Pos3) AND #I_PBSet AND #IO_Modes.LMode.ManualMode AND NOT #IO_Modes.LGeneralFunc.LamptestSteady) OR ((((#CmdPos1 OR #CmdPos2) AND "Blink_0,5s") OR #I_Pos1 OR #I_Pos2) AND #I_PBReset AND #IO_Modes.LMode.ManualMode AND NOT #IO_Modes.LGeneralFunc.LamptestSteady) OR #IO_Modes.LGeneralFunc.Lamptest;
END_REGION

REGION Network 31: **** 8 - Outputs **** Alarm AB Condition
   // Alarm AB Condition
   #O_AlarmABCondition := "FALSE";
END_REGION

REGION Network 32: **** 9 - Alarm Summary **** Alarms To Alarm UDT Alarms To Alarm UDT Get Name
   // Alarm / Alarm D
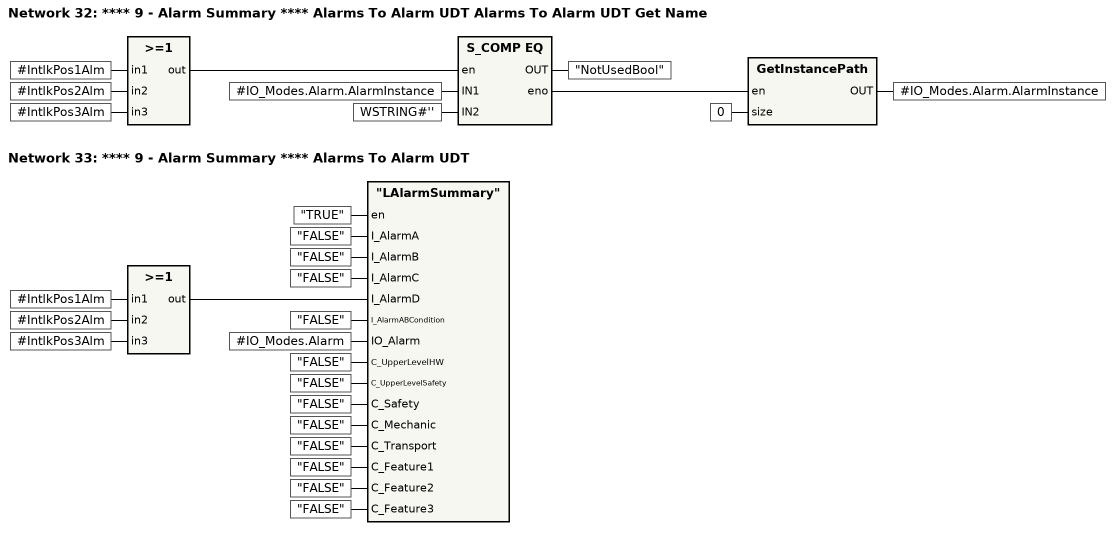
   S_COMP(EN := #IntlkPos1Alm OR #IntlkPos2Alm OR #IntlkPos3Alm,
          IN1 := #IO_Modes.Alarm.AlarmInstance,
          IN2 := WSTRING#'',
          OUT => "NotUsedBool",
          ENO => #_w1);
   IF #_w1 THEN GetInstancePath(size := 0, OUT => #IO_Modes.Alarm.AlarmInstance); END_IF;
END_REGION

REGION Network 33: **** 9 - Alarm Summary **** Alarms To Alarm UDT
   // Alarm / Alarm D
   IF "TRUE" THEN
       "LAlarmSummary"(I_AlarmA := "FALSE",
                       I_AlarmB := "FALSE",
                       I_AlarmC := "FALSE",
                       I_AlarmD := #IntlkPos1Alm OR #IntlkPos2Alm OR #IntlkPos3Alm,
                       I_AlarmABCondition := "FALSE",
                       IO_Alarm := #IO_Modes.Alarm,
                       C_UpperLevelHW := "FALSE",
                       C_UpperLevelSafety := "FALSE",
                       C_Safety := "FALSE",
                       C_Mechanic := "FALSE",
                       C_Transport := "FALSE",
                       C_Feature1 := "FALSE",
                       C_Feature2 := "FALSE",
                       C_Feature3 := "FALSE");
   END_IF;
END_REGION
END_FUNCTION_BLOCK
